FUNCTION_BLOCK TFModulePalletizer_Pinza_mag
VAR_INPUT
	Cmd 	: CommandBuffer;
	Cfg 	: Config;
	IN 		: TFMchinePalletizer_PinzaVentose_IN;
	IN_Ax 	: Module_Palletizer_Ax_IN;
	
	AspirazioneDX1 : POINTER TO TF_VacumOVEM;
	AspirazioneSX1 : POINTER TO TF_VacumOVEM;
	AspirazioneDX2 : POINTER TO TF_VacumOVEM;
	AspirazioneSX2 : POINTER TO TF_VacumOVEM;

	CilindroSbloccoRotazione 	: POINTER TO SC_Cylinder;
	CilindroSbloccoBascolante 	: POINTER TO SC_Cylinder;
	CilindroApertura 			: POINTER TO DC_Cylinder;
	
	ModuleJ : POINTER TO TFModulePalletizer_Ax;
	ModuleK : POINTER TO TFModulePalletizer_Ax;

	ManCmd 				: POINTER TO TFMachinePalletizer_PinzaVentoseManCmd;
	ElementoInPrelievo 	: TFMachinePalletizer_PlaceElement;
	DataElement			: TFMachinePalletizer_DataElement; (* Struttura dati che la macchina acquisisce/trasferisce in fase di pallettizzazione/depallettizazione *)
	PrelievoSuMagazino : BOOL;//indica che il prelievo è su cavallina

	Mission : POINTER TO TFMachinePalletizer_Mission;
	AbilitazioneSbloccoRotazione 	: BOOL;//Abilitazione sblocco rotazione pinza
	AbilitazioneSbloccoBascolante 	: BOOL;//Abilitazione sblocco bascolante pinza	
	IN_SimulazioneSenzaHW : BOOL;
	AbilitaAperturaAutomaticaPinza : BOOL;//Abilitazione apertura automatica pinza
END_VAR
VAR_OUTPUT
	CmdExe 		: CommandExe;
	CmdExd 		: CommandExe;
	CmdNext 	: Command;
	CmdLog 		: CommandLog;
	ProgramLog 	: ProgrammaLog; 
	State 		: State;
	StateLog 	: StateLog;
	Error 		: Error;
	ErrorLog 	: ErrorLog;
	Warning 	: Warning;
	WarningLog	: WarningLog;
	OUT 		: TFMachinePalletizer_PinzaVentose_OUT;
	StatoPinza 	: TFMachinePalletizer_PinzaState;

END_VAR
VAR
	Power 	: UINT;
	Init 	: BOOL;
	Timer 	: REAL;
	Timeout : REAL;
	TimerAspirazione 	: REAL;
	ParametersArray 	: ParametersArray;
	MAN_Actuator 		: UINT;
	MAN_Cmd 			: UINT;

	DistanzaFTC_J0 		: REAL;
	DistanzaFTC_J180 	: REAL;
	DistanzaFTC_K0 		: REAL;
	DistanzaFTC_K180 	: REAL;

	TimerPresaPiastrella : REAL;		
	DisattivazioneTotaleAspirazioni : bool;
	ByPassAttesaDistacco : BOOL;

	DistanzaJForzata : REAL;
	DistanzaKForzata : REAL;

END_VAR

IF NOT Init THEN
	TFCommandBufferClear(ADR(Cmd));
	TFCommandClear(ADR(CmdNext));
	TFCommandExeClear(ADR(CmdExe));
	TFStateUpdate(ADR(State),StateNOP);
	TFErrorClear(ADR(Error));
	TFWarningClear(ADR(Warning));
	Init := TRUE;
END_IF

(* Generic Timer - Add here all your Timers *)
TFTimerCall(ADR(Timer),Cfg.TimeBase);
TFTimerCall(ADR(Timeout),Cfg.TimeBase);
TFTimerCall(ADR(TimerPresaPiastrella),Cfg.TimeBase);
TFTimerCall(ADR(TimerAspirazione),Cfg.TimeBase);
(* External To Buffered Command *)
TFCommandToNext(ADR(Cmd),ADR(CmdNext),ADR(CmdExe),ADR(Cfg),ADR(Error),ADR(ErrorLog),ADR(State));

(* Buffered To Exe Command *)
TFCommandToExecution(ADR(CmdNext),ADR(CmdExe),ADR(Error),ADR(ErrorLog),ADR(State),ADR(CmdLog));

(* Chiamata FB *)
AspirazioneDX1^();
AspirazioneSX1^();
AspirazioneDX2^();
AspirazioneSX2^();
CilindroSbloccoRotazione^();
CilindroSbloccoBascolante^();

DistanzaFTC_J0 		:= Keyence_LRTB2000C(IN.InKeyence_J0_Byte0,IN.InKeyence_J0_Byte1);
DistanzaFTC_J180	:= Keyence_LRTB2000C(IN.InKeyence_J180_Byte0,IN.InKeyence_J180_Byte1);
DistanzaFTC_K0 		:= Keyence_LRTB2000C(IN.InKeyence_K0_Byte0,IN.InKeyence_K0_Byte1);
DistanzaFTC_K180	:= Keyence_LRTB2000C(IN.InKeyence_K180_Byte0,IN.InKeyence_K180_Byte1);

OUT.DistanzaFTC_J0 		:= DistanzaFTC_J0; 		
OUT.DistanzaFTC_J180	:= DistanzaFTC_J180;	
OUT.DistanzaFTC_K0 		:= DistanzaFTC_K0; 		
OUT.DistanzaFTC_K180   	:= DistanzaFTC_K180; 

DistanzaJForzata:=0;
IF ABS(DistanzaFTC_J0-DistanzaFTC_J180) > 30 THEN
	DistanzaJForzata := MIN(DistanzaFTC_J0,DistanzaFTC_J180);
END_IF
DistanzaKForzata:=0;
IF ABS(DistanzaFTC_K0-DistanzaFTC_K180) > 30 THEN
	DistanzaKForzata := MIN(DistanzaFTC_K0,DistanzaFTC_K180);
END_IF
OUT.DistanzaMedia := (DistanzaFTC_J0 + 	
                 DistanzaFTC_J180 +
                 DistanzaFTC_K0 + 	
                 DistanzaFTC_K180)/4;
				 
IF DistanzaKForzata > 0 THEN
	OUT.DistanzaMedia := (DistanzaJForzata +
                 DistanzaFTC_K0 + 	
                 DistanzaFTC_K180)/3;
END_IF
IF DistanzaJForzata > 0 THEN
	OUT.DistanzaMedia := (DistanzaFTC_J0 + 	
                 DistanzaFTC_J180 +
                 DistanzaKForzata)/3;
END_IF
IF DistanzaKForzata > 0 AND DistanzaJForzata > 0 THEN
	OUT.DistanzaMedia := (DistanzaJForzata +
                 DistanzaKForzata)/2;
END_IF

(* Exe Command *)
CASE CmdExe.Code OF

	(* ******************************************************************************************************** *)
	(* Nop  *)
	(* ******************************************************************************************************** *)
	CmdNOP:	;			
	(* ******************************************************************************************************** *)
	(* Stop *)
	(* ******************************************************************************************************** *)
	CmdSTOP:
		CASE CmdExe.CmdCase OF
			
			(* Case 0 *)
			0: 	TFStateUpdate(ADR(State),StateSTOP_RUN);
				TFTimerSet(ADR(Timeout),500,TRUE);
				TFCommandCase(ADR(CmdExe),1,CommandCase_INC);

			(* Case 1 - Clear All Commands*)
			1:	
				TFCommandCase(ADR(CmdExe),100,CommandCase_JMP);
			(* Case 100 *)
			100:TFStateUpdate(ADR(State),StateSTOP_END);
				TFCommandExeClear(ADR(CmdExe));

			ELSE
				TFError(ErrNOCMDCASE,ErrNULL,ADR(CmdExe),ADR(State),ADR(Error),ADR(ErrorLog));
		END_CASE;
	
	(* ******************************************************************************************************** *)
	(* Error Reset *)
	(* ******************************************************************************************************** *)
	CmdRESET:
		CASE CmdExe.CmdCase OF

			(* Case 0 *)
			0: 	TFStateUpdate(ADR(State),StateRESET_RUN);
				TFTimerSet(ADR(Timeout),2000+100,TRUE);
				TFTimerSet(ADR(Timer),2000,TRUE);
				TFCommandCase(ADR(CmdExe),1,CommandCase_JMP);

			
			(* Case 1 - RESET COMANDI*)
			1: 
				TFClearAllCmdModulePinzaMagazzino(AspirazioneDX1,AspirazioneSX1,AspirazioneDX2,AspirazioneSX2,CilindroSbloccoRotazione,CilindroSbloccoBascolante);
				TFCommandCase(ADR(CmdExe),1,CommandCase_INC);
			
			(* Case 2 - Invio comando di reset *)
			2:
				AspirazioneDX1^.Command^.ErrorReset 				:= TRUE;	
				AspirazioneSX1^.Command^.ErrorReset 				:= TRUE;	
				AspirazioneDX2^.Command^.ErrorReset 				:= TRUE;	
				AspirazioneSX2^.Command^.ErrorReset 				:= TRUE;	
				CilindroSbloccoRotazione^.Command.ErrorReset 	:= TRUE;	
				CilindroSbloccoBascolante^.Command.ErrorReset 	:= TRUE;	
				TFCommandCase(ADR(CmdExe),1,CommandCase_INC);
			
			(* Case 3 - Invio comando di reset *)
			3:
				IF (AspirazioneDX1^.Status.ErrorResetDone AND AspirazioneDX2^.Status.ErrorResetDone AND
					AspirazioneSX1^.Status.ErrorResetDone AND AspirazioneSX2^.Status.ErrorResetDone AND
					CilindroSbloccoRotazione^.Status.ErrorResetDone AND CilindroSbloccoBascolante^.Status.ErrorResetDone) OR IN_SimulazioneSenzaHW THEN					
					TFClearAllCmdModulePinzaMagazzino(AspirazioneDX1,AspirazioneSX1,AspirazioneDX2,AspirazioneSX2,CilindroSbloccoRotazione,CilindroSbloccoBascolante);
					TFCommandCase(ADR(CmdExe),99,CommandCase_JMP);
				ELSIF TFTimerDone(ADR(Timer)) THEN
					TFClearAllCmdModulePinzaMagazzino(AspirazioneDX1,AspirazioneSX1,AspirazioneDX2,AspirazioneSX2,CilindroSbloccoRotazione,CilindroSbloccoBascolante);
					TFError(ErrTORESET,ErrNULL,ADR(CmdExe),ADR(State),ADR(Error),ADR(ErrorLog));
				END_IF

			(* Case 99 *)
			99:	TFErrorClear(ADR(Error));
				TFWarningClear(ADR(Warning));
				TFCommandCase(ADR(CmdExe),100,CommandCase_JMP);

			(* Case 100 *)
			100:TFStateUpdate(ADR(State),StateRESET_END);
				TFCommandExeClear(ADR(CmdExe));

			ELSE
				TFError(ErrNOCMDCASE,ErrNULL,ADR(CmdExe),ADR(State),ADR(Error),ADR(ErrorLog));
		END_CASE;

		(*IF AspirazioneDX^.Status.ErrorID <> ErrNULL THEN
			TFClearAllCmdModulePinza(AspirazioneDX,AspirazioneSX,CilindroApertura,CilindroSbloccoRotazione,AspirazioneFaldaDX,AspirazioneFaldaSX,CilindroTasteggio);
			TFError(ErrCYLINDER,AspirazioneDX^.Status.ErrorID,ADR(CmdExe),ADR(State),ADR(Error),ADR(ErrorLog));
		ELSIF AspirazioneSX^.Status.ErrorID <> ErrNULL THEN
			TFClearAllCmdModulePinza(AspirazioneDX,AspirazioneSX,CilindroApertura,CilindroSbloccoRotazione,AspirazioneFaldaDX,AspirazioneFaldaSX,CilindroTasteggio);
			TFError(ErrCYLINDER,AspirazioneSX^.Status.ErrorID,ADR(CmdExe),ADR(State),ADR(Error),ADR(ErrorLog));
		ELSIF CilindroApertura^.Status.ErrorID <> ErrNULL THEN
			TFClearAllCmdModulePinza(AspirazioneDX,AspirazioneSX,CilindroApertura,CilindroSbloccoRotazione,AspirazioneFaldaDX,AspirazioneFaldaSX,CilindroTasteggio);
			TFError(ErrCYLINDER,CilindroApertura^.Status.ErrorID,ADR(CmdExe),ADR(State),ADR(Error),ADR(ErrorLog));
		ELSIF CilindroSbloccoRotazione^.Status.ErrorID <> ErrNULL THEN
			TFClearAllCmdModulePinza(AspirazioneDX,AspirazioneSX,CilindroApertura,CilindroSbloccoRotazione,AspirazioneFaldaDX,AspirazioneFaldaSX,CilindroTasteggio);
			TFError(ErrCYLINDER,CilindroSbloccoRotazione^.Status.ErrorID,ADR(CmdExe),ADR(State),ADR(Error),ADR(ErrorLog));
		ELSIF AspirazioneFaldaDX^.Status.ErrorID <> ErrNULL THEN
			TFClearAllCmdModulePinza(AspirazioneDX,AspirazioneSX,CilindroApertura,CilindroSbloccoRotazione,AspirazioneFaldaDX,AspirazioneFaldaSX,CilindroTasteggio);
			TFError(ErrCYLINDER,AspirazioneFaldaDX^.Status.ErrorID,ADR(CmdExe),ADR(State),ADR(Error),ADR(ErrorLog));
		ELSIF AspirazioneFaldaSX^.Status.ErrorID <> ErrNULL THEN
			TFClearAllCmdModulePinza(AspirazioneDX,AspirazioneSX,CilindroApertura,CilindroSbloccoRotazione,AspirazioneFaldaDX,AspirazioneFaldaSX,CilindroTasteggio);
			TFError(ErrCYLINDER,AspirazioneFaldaSX^.Status.ErrorID,ADR(CmdExe),ADR(State),ADR(Error),ADR(ErrorLog));
		*)
		IF TFTimerDone(ADR(Timeout)) THEN
			TFClearAllCmdModulePinzaMagazzino(AspirazioneDX1,AspirazioneSX1,AspirazioneDX2,AspirazioneSX2,CilindroSbloccoRotazione,CilindroSbloccoBascolante);
			TFError(ErrCMDTIMEOUT,ErrNULL,ADR(CmdExe),ADR(State),ADR(Error),ADR(ErrorLog));
		END_IF
	
	(* ******************************************************************************************************** *)
	(* Power *)
	(* ******************************************************************************************************** *)
	CmdPOWER:
		CASE CmdExe.CmdCase OF
			
			(* Case 0 *)
			0: 	TFStateUpdate(ADR(State),StatePOWER_RUN);
				TFTimerSet(ADR(Timeout),500,TRUE);
				TFCommandCase(ADR(CmdExe),100,CommandCase_JMP);

			1: TFCommandCase(ADR(CmdExe),100,CommandCase_JMP);
			(* Case 100 *)
			100:TFStateUpdate(ADR(State),StatePOWER_END);
				TFCommandExeClear(ADR(CmdExe));

			ELSE
				TFError(ErrNOCMDCASE,ErrNULL,ADR(CmdExe),ADR(State),ADR(Error),ADR(ErrorLog));
		END_CASE
	
	(* ******************************************************************************************************** *)
	(* Home *)
	(* ******************************************************************************************************** *)
	CmdHOME:
		CASE CmdExe.CmdCase OF

			(* Case 0 *)
			0: 	TFStateUpdate(ADR(State),StateHOME_RUN);
				TFTimerSet(ADR(Timeout),3000+200,TRUE);
				TFTimerSet(ADR(Timer),3000,TRUE);
				IF NOT IN_SimulazioneSenzaHW THEN
					TFCommandCase(ADR(CmdExe),1,CommandCase_INC);
				ELSE
					TFCommandCase(ADR(CmdExe),100,CommandCase_JMP);
				END_IF

			(* Case 1 - *)
			1: 
				TFCommandCase(ADR(CmdExe),10,CommandCase_JMP);

			(* Case 10 - Set automatico Soglie *)
			10:
				AspirazioneDX1^.Command^.Aspirazione_ON_ScritturaSoglia 	:= TRUE;
				AspirazioneSX1^.Command^.Aspirazione_ON_ScritturaSoglia 	:= TRUE;
				AspirazioneDX2^.Command^.Aspirazione_ON_ScritturaSoglia 	:= TRUE;
				AspirazioneSX2^.Command^.Aspirazione_ON_ScritturaSoglia 	:= TRUE;
				IF AspirazioneDX1^.Status.CommandDone AND AspirazioneSX1^.Status.CommandDone AND
					AspirazioneDX2^.Status.CommandDone AND AspirazioneSX2^.Status.CommandDone THEN
						TFClearAllCmdModulePinzaMagazzino(AspirazioneDX1,AspirazioneSX1,AspirazioneDX2,AspirazioneSX2,CilindroSbloccoRotazione,CilindroSbloccoBascolante);
						TFCommandCase(ADR(CmdExe),100,CommandCase_JMP);
				ELSIF TFTimerDone(ADR(Timer)) THEN
					TFClearAllCmdModulePinzaMagazzino(AspirazioneDX1,AspirazioneSX1,AspirazioneDX2,AspirazioneSX2,CilindroSbloccoRotazione,CilindroSbloccoBascolante);
					TFError(ErrTOHOME,ErrNULL,ADR(CmdExe),ADR(State),ADR(Error),ADR(ErrorLog));
				END_IF
			
	
			(* Case 100 *)
			100:TFStateUpdate(ADR(State),StateHOME_END);
				TFCommandExeClear(ADR(CmdExe));

			ELSE
				TFError(ErrNOCMDCASE,ErrNULL,ADR(CmdExe),ADR(State),ADR(Error),ADR(ErrorLog));
		END_CASE;
		
		IF AspirazioneDX1^.Status.ErrorID <> ErrNULL AND NOT IN_SimulazioneSenzaHW THEN
			TFClearAllCmdModulePinzaMagazzino(AspirazioneDX1,AspirazioneSX1,AspirazioneDX2,AspirazioneSX2,CilindroSbloccoRotazione,CilindroSbloccoBascolante);
			TFError(ErrCYLINDER,AspirazioneDX1^.Status.ErrorID,ADR(CmdExe),ADR(State),ADR(Error),ADR(ErrorLog));
		ELSIF AspirazioneSX1^.Status.ErrorID <> ErrNULL AND NOT IN_SimulazioneSenzaHW THEN
			TFClearAllCmdModulePinzaMagazzino(AspirazioneDX1,AspirazioneSX1,AspirazioneDX2,AspirazioneSX2,CilindroSbloccoRotazione,CilindroSbloccoBascolante);
			TFError(ErrCYLINDER,AspirazioneSX1^.Status.ErrorID,ADR(CmdExe),ADR(State),ADR(Error),ADR(ErrorLog));
		ELSIF AspirazioneDX2^.Status.ErrorID <> ErrNULL AND NOT IN_SimulazioneSenzaHW THEN
			TFClearAllCmdModulePinzaMagazzino(AspirazioneDX1,AspirazioneSX1,AspirazioneDX2,AspirazioneSX2,CilindroSbloccoRotazione,CilindroSbloccoBascolante);
			TFError(ErrCYLINDER,AspirazioneDX2^.Status.ErrorID,ADR(CmdExe),ADR(State),ADR(Error),ADR(ErrorLog));
		ELSIF AspirazioneSX2^.Status.ErrorID <> ErrNULL AND NOT IN_SimulazioneSenzaHW THEN
			TFClearAllCmdModulePinzaMagazzino(AspirazioneDX1,AspirazioneSX1,AspirazioneDX2,AspirazioneSX2,CilindroSbloccoRotazione,CilindroSbloccoBascolante);
			TFError(ErrCYLINDER,AspirazioneSX2^.Status.ErrorID,ADR(CmdExe),ADR(State),ADR(Error),ADR(ErrorLog));
		ELSIF CilindroSbloccoRotazione^.Status.ErrorID <> ErrNULL THEN
			TFClearAllCmdModulePinzaMagazzino(AspirazioneDX1,AspirazioneSX1,AspirazioneDX2,AspirazioneSX2,CilindroSbloccoRotazione,CilindroSbloccoBascolante);
			TFError(ErrCYLINDER,CilindroSbloccoRotazione^.Status.ErrorID,ADR(CmdExe),ADR(State),ADR(Error),ADR(ErrorLog));
		ELSIF TFTimerDone(ADR(Timeout)) THEN
			TFClearAllCmdModulePinzaMagazzino(AspirazioneDX1,AspirazioneSX1,AspirazioneDX2,AspirazioneSX2,CilindroSbloccoRotazione,CilindroSbloccoBascolante);
			TFError(ErrCMDTIMEOUT,ErrNULL,ADR(CmdExe),ADR(State),ADR(Error),ADR(ErrorLog));
		END_IF

	(* ******************************************************************************************************** *)
	(* Manual *)
	(* ******************************************************************************************************** *)
	CmdMAN:
		CASE CmdExe.CmdCase OF
			(* Case 0 *)
			0: 	TFStateUpdate(ADR(State),StateMAN_RUN);
				TFTimerSet(ADR(Timeout),3000,TRUE);
				TFTimerSet(ADR(Timer),10,TRUE);
				IF TFCommandParRead(CmdExe.Cmd.Parameter,ADR(ParametersArray),2) THEN
					MAN_Actuator	:= STRING_TO_UINT(ParametersArray.Parameters[0]);
					MAN_Cmd		:= STRING_TO_UINT(ParametersArray.Parameters[1]);
				ELSE
					TFError(ErrCMDPARNUM,ErrNULL,ADR(CmdExe),ADR(State),ADR(Error),ADR(ErrorLog));
					RETURN;
				END_IF;

				CASE MAN_Actuator OF
					(* Case 0..99 for Actuators *)
					(* Case 100..199  for Axis *)

					(* Case Nop *)
					0:	;

					(* Case 1: *)
					1:	CASE MAN_Cmd OF
							0:	;
							
							
							(* Case 20: Sgancio Sblocco Rotazione *)
							20:	
								CilindroSbloccoRotazione^.Command.Activation 	:= TRUE;
								CilindroSbloccoRotazione^.Command.Deactivation 	:= FALSE;
								TFTimerSet(ADR(Timeout),3000,TRUE);
								TFCommandCase(ADR(CmdExe),20,CommandCase_JMP);
								
							(* Case 21: Aggancio Sblocco Rotazione *)
							21:	
								CilindroSbloccoRotazione^.Command.Activation 	:= FALSE;
								CilindroSbloccoRotazione^.Command.Deactivation 	:= TRUE;
								TFTimerSet(ADR(Timeout),3000,TRUE);
								TFCommandCase(ADR(CmdExe),20,CommandCase_JMP);
	
							(* Case 50: Ativazione Aspirazione SX *)
							50:	
								
								IF NOT IN_SimulazioneSenzaHW THEN 
									AspirazioneSX1^.Command^.Aspirazione_ON		:= TRUE;
									AspirazioneSX1^.Command^.Aspirazione_OFF 	:= FALSE;
									AspirazioneDX1^.Command^.Aspirazione_ON 	:= TRUE;
									AspirazioneDX1^.Command^.Aspirazione_OFF 	:= FALSE;
									AspirazioneSX2^.Command^.Aspirazione_ON 	:= TRUE;
									AspirazioneSX2^.Command^.Aspirazione_OFF 	:= FALSE;
									AspirazioneDX2^.Command^.Aspirazione_ON 	:= TRUE;
									AspirazioneDX2^.Command^.Aspirazione_OFF 	:= FALSE;
	
									TFTimerSet(ADR(Timeout),3000,TRUE);
									TFCommandCase(ADR(CmdExe),50,CommandCase_JMP);
								ELSE
									TFCommandCase(ADR(CmdExe),1,CommandCase_JMP);
								END_IF
										
							(* Case 51: Disattivazione Aspirazione SX *)
							51:	
								StatoPinza.ElementoPrelevato := FALSE;
								IF NOT IN_SimulazioneSenzaHW THEN 
									AspirazioneSX1^.Command^.Aspirazione_ON 	:= FALSE;
									AspirazioneSX1^.Command^.Aspirazione_OFF 	:= TRUE;
									AspirazioneDX1^.Command^.Aspirazione_ON 	:= FALSE;
									AspirazioneDX1^.Command^.Aspirazione_OFF 	:= TRUE;
									AspirazioneSX2^.Command^.Aspirazione_ON 	:= FALSE;
									AspirazioneSX2^.Command^.Aspirazione_OFF 	:= TRUE;
									AspirazioneDX2^.Command^.Aspirazione_ON 	:= FALSE;
									AspirazioneDX2^.Command^.Aspirazione_OFF 	:= TRUE;
									TFTimerSet(ADR(Timeout),3000,TRUE);
									TFCommandCase(ADR(CmdExe),50,CommandCase_JMP);
								ELSE
									TFCommandCase(ADR(CmdExe),1,CommandCase_JMP);
								END_IF

							(* Case 60: Ativazione Aspirazione DX *)
							60:	
								IF NOT IN_SimulazioneSenzaHW THEN 
									AspirazioneSX1^.Command^.Aspirazione_ON 	:= TRUE;
									AspirazioneSX1^.Command^.Aspirazione_OFF 	:= FALSE;
									AspirazioneDX1^.Command^.Aspirazione_ON 	:= TRUE;
									AspirazioneDX1^.Command^.Aspirazione_OFF 	:= FALSE;
									AspirazioneSX2^.Command^.Aspirazione_ON 	:= TRUE;
									AspirazioneSX2^.Command^.Aspirazione_OFF 	:= FALSE;
									AspirazioneDX2^.Command^.Aspirazione_ON 	:= TRUE;
									AspirazioneDX2^.Command^.Aspirazione_OFF 	:= FALSE;
									TFTimerSet(ADR(Timeout),3000,TRUE);
									TFCommandCase(ADR(CmdExe),60,CommandCase_JMP);
								ELSE
									TFCommandCase(ADR(CmdExe),1,CommandCase_JMP);
								END_IF

							(* Case 61: Disattivazione Aspirazione SX *)
							61:	
								StatoPinza.ElementoPrelevato := FALSE;
								IF NOT IN_SimulazioneSenzaHW THEN 
									AspirazioneDX1^.Command^.Aspirazione_ON  := FALSE;
									AspirazioneDX1^.Command^.Aspirazione_OFF := TRUE;
									AspirazioneSX1^.Command^.Aspirazione_ON  := FALSE;
									AspirazioneSX1^.Command^.Aspirazione_OFF := TRUE;
									AspirazioneDX2^.Command^.Aspirazione_ON  := FALSE;
									AspirazioneDX2^.Command^.Aspirazione_OFF := TRUE;
									AspirazioneSX2^.Command^.Aspirazione_ON  := FALSE;
									AspirazioneSX2^.Command^.Aspirazione_OFF := TRUE;
									StatoPinza.ElementoPrelevato := FALSE;
									TFTimerSet(ADR(Timeout),3000,TRUE);
									TFCommandCase(ADR(CmdExe),60,CommandCase_JMP);
								ELSE
									TFCommandCase(ADR(CmdExe),1,CommandCase_JMP);
								END_IF
							ELSE
								TFError(ErrNOCMDCASE,ErrNULL,ADR(CmdExe),ADR(State),ADR(Error),ADR(ErrorLog));
						END_CASE;

					100:CASE MAN_Cmd OF
							0:	;
							ELSE
								TFError(ErrNOCMDCASE,ErrNULL,ADR(CmdExe),ADR(State),ADR(Error),ADR(ErrorLog));
						END_CASE;

					ELSE
						TFError(ErrNOCMDCASE,ErrNULL,ADR(CmdExe),ADR(State),ADR(Error),ADR(ErrorLog));
				END_CASE;

				//IF CmdExe.CmdCase = 0 THEN
					//TFCommandCase(ADR(CmdExe),1,CommandCase_INC);
				//END_IF

			(* Case 1 - *)
			1: 	IF (MAN_Cmd = 0) OR TFTimerDone(ADR(Timer)) THEN
					(* Clear All Output Here *)
					;
					TFStateUpdate(ADR(State),StateMAN_END);
					TFCommandExeClear(ADR(CmdExe));
				END_IF;

			(* Case 20 - CilindroSbloccoRotazione *)
			20: 
				IF CilindroSbloccoRotazione^.Status.Inactive AND CilindroSbloccoRotazione^.Command.Deactivation OR
					CilindroSbloccoRotazione^.Status.Active AND CilindroSbloccoRotazione^.Command.Activation THEN
						CilindroSbloccoRotazione^.Command.Activation 	:= FALSE;
						CilindroSbloccoRotazione^.Command.Deactivation 	:= FALSE;
						TFCommandCase(ADR(CmdExe),100,CommandCase_JMP);
				ELSIF CilindroSbloccoRotazione^.Status.ErrorID <> ErrNULL THEN
					TFClearAllCmdModulePinzaMagazzino(AspirazioneDX1,AspirazioneSX1,AspirazioneDX2,AspirazioneSX2,CilindroSbloccoRotazione,CilindroSbloccoBascolante);
					TFError(ErrCYLINDER,CilindroSbloccoRotazione^.Status.ErrorID,ADR(CmdExe),ADR(State),ADR(Error),ADR(ErrorLog));
				END_IF

			(* Case 50 - AspirazioneSX *)
			50: 
				IF AspirazioneSX1^.Status.CommandDone AND AspirazioneDX1^.Status.CommandDone AND
					AspirazioneSX2^.Status.CommandDone AND AspirazioneDX2^.Status.CommandDone THEN
						TFClearAllCmdModulePinzaMagazzino(AspirazioneDX1,AspirazioneSX1,AspirazioneDX2,AspirazioneSX2,CilindroSbloccoRotazione,CilindroSbloccoBascolante);
						TFCommandCase(ADR(CmdExe),100,CommandCase_JMP);
				ELSIF AspirazioneSX1^.Status.ErrorID <> ErrNULL THEN
					TFClearAllCmdModulePinzaMagazzino(AspirazioneDX1,AspirazioneSX1,AspirazioneDX2,AspirazioneSX2,CilindroSbloccoRotazione,CilindroSbloccoBascolante);
					TFError(ErrCYLINDER,AspirazioneSX1^.Status.ErrorID,ADR(CmdExe),ADR(State),ADR(Error),ADR(ErrorLog));
				ELSIF AspirazioneDX1^.Status.ErrorID <> ErrNULL THEN
					TFClearAllCmdModulePinzaMagazzino(AspirazioneDX1,AspirazioneSX1,AspirazioneDX2,AspirazioneSX2,CilindroSbloccoRotazione,CilindroSbloccoBascolante);
					TFError(ErrCYLINDER,AspirazioneDX1^.Status.ErrorID,ADR(CmdExe),ADR(State),ADR(Error),ADR(ErrorLog));
				ELSIF AspirazioneSX2^.Status.ErrorID <> ErrNULL THEN
					TFClearAllCmdModulePinzaMagazzino(AspirazioneDX1,AspirazioneSX1,AspirazioneDX2,AspirazioneSX2,CilindroSbloccoRotazione,CilindroSbloccoBascolante);
					TFError(ErrCYLINDER,AspirazioneSX2^.Status.ErrorID,ADR(CmdExe),ADR(State),ADR(Error),ADR(ErrorLog));
				ELSIF AspirazioneDX2^.Status.ErrorID <> ErrNULL THEN
					TFClearAllCmdModulePinzaMagazzino(AspirazioneDX1,AspirazioneSX1,AspirazioneDX2,AspirazioneSX2,CilindroSbloccoRotazione,CilindroSbloccoBascolante);
					TFError(ErrCYLINDER,AspirazioneDX2^.Status.ErrorID,ADR(CmdExe),ADR(State),ADR(Error),ADR(ErrorLog));
				END_IF

			(* Case 60 - AspirazioneDX *)
			60: 
				IF AspirazioneSX1^.Status.CommandDone AND AspirazioneDX1^.Status.CommandDone AND
					AspirazioneSX2^.Status.CommandDone AND AspirazioneDX2^.Status.CommandDone THEN
						TFClearAllCmdModulePinzaMagazzino(AspirazioneDX1,AspirazioneSX1,AspirazioneDX2,AspirazioneSX2,CilindroSbloccoRotazione,CilindroSbloccoBascolante);
						TFCommandCase(ADR(CmdExe),100,CommandCase_JMP);
				ELSIF AspirazioneSX1^.Status.ErrorID <> ErrNULL THEN
					TFClearAllCmdModulePinzaMagazzino(AspirazioneDX1,AspirazioneSX1,AspirazioneDX2,AspirazioneSX2,CilindroSbloccoRotazione,CilindroSbloccoBascolante);
					TFError(ErrCYLINDER,AspirazioneSX1^.Status.ErrorID,ADR(CmdExe),ADR(State),ADR(Error),ADR(ErrorLog));
				ELSIF AspirazioneDX1^.Status.ErrorID <> ErrNULL THEN
					TFClearAllCmdModulePinzaMagazzino(AspirazioneDX1,AspirazioneSX1,AspirazioneDX2,AspirazioneSX2,CilindroSbloccoRotazione,CilindroSbloccoBascolante);
					TFError(ErrCYLINDER,AspirazioneDX1^.Status.ErrorID,ADR(CmdExe),ADR(State),ADR(Error),ADR(ErrorLog));
				ELSIF AspirazioneSX2^.Status.ErrorID <> ErrNULL THEN
					TFClearAllCmdModulePinzaMagazzino(AspirazioneDX1,AspirazioneSX1,AspirazioneDX2,AspirazioneSX2,CilindroSbloccoRotazione,CilindroSbloccoBascolante);
					TFError(ErrCYLINDER,AspirazioneSX2^.Status.ErrorID,ADR(CmdExe),ADR(State),ADR(Error),ADR(ErrorLog));
				ELSIF AspirazioneDX2^.Status.ErrorID <> ErrNULL THEN
					TFClearAllCmdModulePinzaMagazzino(AspirazioneDX1,AspirazioneSX1,AspirazioneDX2,AspirazioneSX2,CilindroSbloccoRotazione,CilindroSbloccoBascolante);
					TFError(ErrCYLINDER,AspirazioneDX2^.Status.ErrorID,ADR(CmdExe),ADR(State),ADR(Error),ADR(ErrorLog));
				END_IF

			(* Case 100 - End *)
			100:(* Clear All Output Here *)
				TFStateUpdate(ADR(State),StateMAN_END);
				TFCommandExeClear(ADR(CmdExe));

			ELSE
				TFError(ErrNOCMDCASE,ErrNULL,ADR(CmdExe),ADR(State),ADR(Error),ADR(ErrorLog));
		END_CASE;

		IF TFTimerDone(ADR(Timeout)) THEN
			TFClearAllCmdModulePinzaMagazzino(AspirazioneDX1,AspirazioneSX1,AspirazioneDX2,AspirazioneSX2,CilindroSbloccoRotazione,CilindroSbloccoBascolante);
			TFError(ErrCMDTIMEOUT,ErrNULL,ADR(CmdExe),ADR(State),ADR(Error),ADR(ErrorLog));
		END_IF
	

	(* ******************************************************************************************************** *)
	(* PRELOAD - Attivazione vuoto *)
	(* ******************************************************************************************************** *)
	CmdPRELOAD:
		CASE CmdExe.CmdCase OF
			
			(* Case 0 - Init Command*)
			0: 	TFStateUpdate(ADR(State),StatePRELOAD_RUN);
				TFTimerSet(ADR(Timeout),30000+200,TRUE);
				TFTimerSet(ADR(Timer),30000,TRUE);
				PrelievoSuMagazino := FALSE;
				StatoPinza.ElementoPrelevato := FALSE;
				IF TFCommandParRead(CmdExe.Cmd.Parameter,ADR(ParametersArray),1) THEN
					PrelievoSuMagazino	:= STRING_TO_BOOL(ParametersArray.Parameters[0]);
					IF NOT IN_SimulazioneSenzaHW THEN
						TFCommandCase(ADR(CmdExe),40,CommandCase_JMP);
					ELSE
						TFCommandCase(ADR(CmdExe),100,CommandCase_JMP);
					END_IF
				ELSE
					TFError(ErrCMDPARNUM,ErrNULL,ADR(CmdExe),ADR(State),ADR(Error),ADR(ErrorLog));
					RETURN;
				END_IF;
				
			(* Case 10 - CilindroSbloccoRotazione *)
			10: 
				IF PrelievoSuMagazino AND FALSE THEN
					CilindroSbloccoRotazione^.Command.Activation 	:= AbilitazioneSbloccoRotazione;
					CilindroSbloccoRotazione^.Command.Deactivation 	:= FALSE;
	
					IF (CilindroSbloccoRotazione^.Status.Active OR NOT AbilitazioneSbloccoRotazione)THEN
						CilindroSbloccoRotazione^.Command.Activation 	:= FALSE;
						CilindroSbloccoRotazione^.Command.Deactivation 	:= FALSE;
						TFCommandCase(ADR(CmdExe),40,CommandCase_JMP);
					ELSIF CilindroSbloccoRotazione^.Status.ErrorID <> ErrNULL AND AbilitazioneSbloccoRotazione THEN
						TFClearAllCmdModulePinzaMagazzino(AspirazioneDX1,AspirazioneSX1,AspirazioneDX2,AspirazioneSX2,CilindroSbloccoRotazione,CilindroSbloccoBascolante);
						TFError(ErrCYLINDER,CilindroSbloccoRotazione^.Status.ErrorID,ADR(CmdExe),ADR(State),ADR(Error),ADR(ErrorLog));
					END_IF
				ELSE
					TFCommandCase(ADR(CmdExe),40,CommandCase_JMP);
				END_IF


			(* Case 40 - AspirazioneDX + AspirazioneSX *)
			40: 
				AspirazioneDX1^.Command^.Aspirazione_ON 	:= TRUE;
				AspirazioneDX1^.Command^.Aspirazione_OFF 	:= FALSE;
				AspirazioneSX1^.Command^.Aspirazione_ON 	:= TRUE;
				AspirazioneSX1^.Command^.Aspirazione_OFF 	:= FALSE;
				AspirazioneDX2^.Command^.Aspirazione_ON 	:= TRUE;
				AspirazioneDX2^.Command^.Aspirazione_OFF 	:= FALSE;
				AspirazioneSX2^.Command^.Aspirazione_ON 	:= TRUE;
				AspirazioneSX2^.Command^.Aspirazione_OFF 	:= FALSE;
	
				IF (AspirazioneDX1^.Status.CommandDone AND AspirazioneSX1^.Status.CommandDone AND
					AspirazioneDX2^.Status.CommandDone AND AspirazioneSX2^.Status.CommandDone) OR IN.ByPassSensoreVuoto THEN
						TFClearAllCmdModulePinzaMagazzino(AspirazioneDX1,AspirazioneSX1,AspirazioneDX2,AspirazioneSX2,CilindroSbloccoRotazione,CilindroSbloccoBascolante);
						TFCommandCase(ADR(CmdExe),100,CommandCase_JMP);
				ELSIF AspirazioneSX1^.Status.ErrorID <> ErrNULL AND NOT IN_SimulazioneSenzaHW THEN
					TFClearAllCmdModulePinzaMagazzino(AspirazioneDX1,AspirazioneSX1,AspirazioneDX2,AspirazioneSX2,CilindroSbloccoRotazione,CilindroSbloccoBascolante);
					TFError(ErrCYLINDER,AspirazioneSX1^.Status.ErrorID,ADR(CmdExe),ADR(State),ADR(Error),ADR(ErrorLog));
				ELSIF AspirazioneDX1^.Status.ErrorID <> ErrNULL AND NOT IN_SimulazioneSenzaHW THEN
					TFClearAllCmdModulePinzaMagazzino(AspirazioneDX1,AspirazioneSX1,AspirazioneDX2,AspirazioneSX2,CilindroSbloccoRotazione,CilindroSbloccoBascolante);
					TFError(ErrCYLINDER,AspirazioneDX1^.Status.ErrorID,ADR(CmdExe),ADR(State),ADR(Error),ADR(ErrorLog));
				ELSIF AspirazioneSX2^.Status.ErrorID <> ErrNULL THEN
					TFClearAllCmdModulePinzaMagazzino(AspirazioneDX1,AspirazioneSX1,AspirazioneDX2,AspirazioneSX2,CilindroSbloccoRotazione,CilindroSbloccoBascolante);
					TFError(ErrCYLINDER,AspirazioneSX2^.Status.ErrorID,ADR(CmdExe),ADR(State),ADR(Error),ADR(ErrorLog));
				ELSIF AspirazioneDX2^.Status.ErrorID <> ErrNULL THEN
					TFClearAllCmdModulePinzaMagazzino(AspirazioneDX1,AspirazioneSX1,AspirazioneDX2,AspirazioneSX2,CilindroSbloccoRotazione,CilindroSbloccoBascolante);
					TFError(ErrCYLINDER,AspirazioneDX2^.Status.ErrorID,ADR(CmdExe),ADR(State),ADR(Error),ADR(ErrorLog));
				END_IF
				
			(* Case 100 *)
			100:TFStateUpdate(ADR(State),StatePRELOAD_END);
				TFCommandExeClear(ADR(CmdExe));

			ELSE
				TFError(ErrNOCMDCASE,ErrNULL,ADR(CmdExe),ADR(State),ADR(Error),ADR(ErrorLog));
		END_CASE

		IF TFTimerDone(ADR(Timeout)) THEN
			TFClearAllCmdModulePinzaMagazzino(AspirazioneDX1,AspirazioneSX1,AspirazioneDX2,AspirazioneSX2,CilindroSbloccoRotazione,CilindroSbloccoBascolante);
			TFError(ErrCMDTIMEOUT,ErrNULL,ADR(CmdExe),ADR(State),ADR(Error),ADR(ErrorLog));
		END_IF
	
	(* ******************************************************************************************************** *)
	(* LOAD - Presa del pezzo *)
	(* ******************************************************************************************************** *)
	CmdCHECKPRESENCE:
		CASE CmdExe.CmdCase OF
			
			(* Case 0 - Init Command*)
			0: 	TFStateUpdate(ADR(State),StateCHECKPRESENCE_RUN);
				TFTimerSet(ADR(Timeout),60000.0+100+HMI_TempoControlloPresaPiastrella,TRUE);
				TFTimerSet(ADR(Timer),2000.0+HMI_TempoControlloPresaPiastrella,TRUE);
				TFTimerSet(ADR(TimerPresaPiastrella),HMI_TempoControlloPresaPiastrella,TRUE);
				StatoPinza.ElementoPrelevato := FALSE;

				TFCommandCase(ADR(CmdExe),1,CommandCase_INC);
				
			(* Case 1 - *)					
			1:
				IF IN.ByPassSensoreVuoto OR TFTimerDone(ADR(TimerPresaPiastrella)) THEN 
					//Tutte piastrelle o tutte falde
					IF (AspirazioneDX1^.Status.DepressioneSoglia1_OK AND AspirazioneSX1^.Status.DepressioneSoglia1_OK AND
						 AspirazioneDX2^.Status.DepressioneSoglia1_OK AND AspirazioneSX2^.Status.DepressioneSoglia1_OK) OR IN.ByPassSensoreVuoto THEN
						StatoPinza.ElementoPrelevato := TRUE;
						TFCommandCase(ADR(CmdExe),11,CommandCase_JMP);
					ELSIF TFTimerDone(ADR(TimerPresaPiastrella)) THEN
						TFCommandCase(ADR(CmdExe),11,CommandCase_JMP);
						StatoPinza.ElementoPrelevato := IN.ByPassSensoreVuoto;	
					END_IF			
				END_IF
				IF TFTimerDone(ADR(Timer)) THEN
					TFClearAllCmdModulePinzaMagazzino(AspirazioneDX1,AspirazioneSX1,AspirazioneDX2,AspirazioneSX2,CilindroSbloccoRotazione,CilindroSbloccoBascolante);
					TFError(ErrMalfunzionamentoSensoriPresenzaPinza,ErrNULL,ADR(CmdExe),ADR(State),ADR(Error),ADR(ErrorLog));
				ELSIF TFTimerDone(ADR(Timeout)) THEN
					TFClearAllCmdModulePinzaMagazzino(AspirazioneDX1,AspirazioneSX1,AspirazioneDX2,AspirazioneSX2,CilindroSbloccoRotazione,CilindroSbloccoBascolante);
					TFError(ErrCMDTIMEOUT,ErrNULL,ADR(CmdExe),ADR(State),ADR(Error),ADR(ErrorLog));
				END_IF
						
			(* Case 11 - *)		
			11:
				TFStateUpdate(ADR(State),StateCHECKPRESENCE_RUN+10);
				TFCommandCase(ADR(CmdExe),100,CommandCase_JMP);
								
					
			(* Case 100 *)
			100:TFStateUpdate(ADR(State),StateCHECKPRESENCE_END);
				TFCommandExeClear(ADR(CmdExe));

			ELSE
				TFError(ErrNOCMDCASE,ErrNULL,ADR(CmdExe),ADR(State),ADR(Error),ADR(ErrorLog));
		END_CASE

	(* ******************************************************************************************************** *)
	(* CmdSbloccaBascolante - SGANCIO BASCULANTE *)
	(* ******************************************************************************************************** *)
	CmdSbloccaBascolante:
		CASE CmdExe.CmdCase OF
			
			(* Case 0 - Init Command*)
			0: 	TFStateUpdate(ADR(State),StateSbloccaBascolante_RUN);
				TFTimerSet(ADR(Timeout),30000+200,TRUE);
				TFTimerSet(ADR(Timer),30000,TRUE);
				IF NOT IN_SimulazioneSenzaHW THEN
					TFCommandCase(ADR(CmdExe),10,CommandCase_JMP);
				ELSE
					TFCommandCase(ADR(CmdExe),100,CommandCase_JMP);
				END_IF
				
			(* Case 10 - CilindroSblocco bacolante *)
			10: 
				CilindroSbloccoBascolante^.Command.Activation 	:= AbilitazioneSbloccoBascolante;
				CilindroSbloccoBascolante^.Command.Deactivation := FALSE;

				IF (CilindroSbloccoBascolante^.Status.Active OR NOT AbilitazioneSbloccoBascolante)THEN
					CilindroSbloccoBascolante^.Command.Activation 	:= FALSE;
					CilindroSbloccoBascolante^.Command.Deactivation 	:= FALSE;
					TFCommandCase(ADR(CmdExe),100,CommandCase_JMP);
				ELSIF CilindroSbloccoBascolante^.Status.ErrorID <> ErrNULL AND AbilitazioneSbloccoBascolante THEN
					TFClearAllCmdModulePinzaMagazzino(AspirazioneDX1,AspirazioneSX1,AspirazioneDX2,AspirazioneSX2,CilindroSbloccoRotazione,CilindroSbloccoBascolante);
					TFError(ErrCYLINDER,CilindroSbloccoBascolante^.Status.ErrorID,ADR(CmdExe),ADR(State),ADR(Error),ADR(ErrorLog));
				END_IF

				
			(* Case 100 *)
			100:TFStateUpdate(ADR(State),StateSbloccaBascolante_END);
				TFCommandExeClear(ADR(CmdExe));

			ELSE
				TFError(ErrNOCMDCASE,ErrNULL,ADR(CmdExe),ADR(State),ADR(Error),ADR(ErrorLog));
		END_CASE

		IF TFTimerDone(ADR(Timeout)) THEN
			TFClearAllCmdModulePinzaMagazzino(AspirazioneDX1,AspirazioneSX1,AspirazioneDX2,AspirazioneSX2,CilindroSbloccoRotazione,CilindroSbloccoBascolante);
			TFError(ErrCMDTIMEOUT,ErrNULL,ADR(CmdExe),ADR(State),ADR(Error),ADR(ErrorLog));
		END_IF
		
		(* ******************************************************************************************************** *)
	(* CmdBloccaBascolante - AGGANCIO BASCULANTE *)
	(* ******************************************************************************************************** *)
	CmdBloccaBascolante:
		CASE CmdExe.CmdCase OF
			
			(* Case 0 - Init Command*)
			0: 	TFStateUpdate(ADR(State),StateBloccaBascolante_RUN);
				TFTimerSet(ADR(Timeout),30000+200,TRUE);
				TFTimerSet(ADR(Timer),30000,TRUE);
				IF NOT IN_SimulazioneSenzaHW THEN
					TFCommandCase(ADR(CmdExe),10,CommandCase_JMP);
				ELSE
					TFCommandCase(ADR(CmdExe),100,CommandCase_JMP);
				END_IF
				
			(* Case 10 - CilindroSblocco bacolante *)
			10: 
				CilindroSbloccoBascolante^.Command.Activation 	:= FALSE;
				CilindroSbloccoBascolante^.Command.Deactivation := TRUE;

				IF  CilindroSbloccoBascolante^.Status.Inactive THEN
					CilindroSbloccoBascolante^.Command.Activation 	:= FALSE;
					CilindroSbloccoBascolante^.Command.Deactivation := FALSE;
					TFCommandCase(ADR(CmdExe),100,CommandCase_JMP);
				ELSIF CilindroSbloccoBascolante^.Status.ErrorID <> ErrNULL AND AbilitazioneSbloccoBascolante THEN
					TFClearAllCmdModulePinzaMagazzino(AspirazioneDX1,AspirazioneSX1,AspirazioneDX2,AspirazioneSX2,CilindroSbloccoRotazione,CilindroSbloccoBascolante);
					TFError(ErrCYLINDER,CilindroSbloccoBascolante^.Status.ErrorID,ADR(CmdExe),ADR(State),ADR(Error),ADR(ErrorLog));
				END_IF

				
			(* Case 100 *)
			100:TFStateUpdate(ADR(State),StateBloccaBascolante_END);
				TFCommandExeClear(ADR(CmdExe));

			ELSE
				TFError(ErrNOCMDCASE,ErrNULL,ADR(CmdExe),ADR(State),ADR(Error),ADR(ErrorLog));
		END_CASE

		IF TFTimerDone(ADR(Timeout)) THEN
			TFClearAllCmdModulePinzaMagazzino(AspirazioneDX1,AspirazioneSX1,AspirazioneDX2,AspirazioneSX2,CilindroSbloccoRotazione,CilindroSbloccoBascolante);
			TFError(ErrCMDTIMEOUT,ErrNULL,ADR(CmdExe),ADR(State),ADR(Error),ADR(ErrorLog));
		END_IF
		
	(* ******************************************************************************************************** *)
	(* CmdSbloccaRotazione - SGANCIO rotazione *)
	(* ******************************************************************************************************** *)
	CmdSbloccaRotazione:
		CASE CmdExe.CmdCase OF
			
			(* Case 0 - Init Command*)
			0: 	TFStateUpdate(ADR(State),StateSbloccaRotazione_RUN);
				TFTimerSet(ADR(Timeout),30000+200,TRUE);
				TFTimerSet(ADR(Timer),30000,TRUE);
				IF NOT IN_SimulazioneSenzaHW THEN
					TFCommandCase(ADR(CmdExe),10,CommandCase_JMP);
				ELSE
					TFCommandCase(ADR(CmdExe),100,CommandCase_JMP);
				END_IF
				
			(* Case 10 - CilindroSblocco bacolante *)
			10: 
				CilindroSbloccoRotazione^.Command.Activation 	:= AbilitazioneSbloccoRotazione;
				CilindroSbloccoRotazione^.Command.Deactivation := FALSE;

				IF (CilindroSbloccoRotazione^.Status.Active OR NOT AbilitazioneSbloccoRotazione)THEN
					CilindroSbloccoRotazione^.Command.Activation 	:= FALSE;
					CilindroSbloccoRotazione^.Command.Deactivation 	:= FALSE;
					TFCommandCase(ADR(CmdExe),100,CommandCase_JMP);
				ELSIF CilindroSbloccoBascolante^.Status.ErrorID <> ErrNULL AND AbilitazioneSbloccoRotazione THEN
					TFClearAllCmdModulePinzaMagazzino(AspirazioneDX1,AspirazioneSX1,AspirazioneDX2,AspirazioneSX2,CilindroSbloccoRotazione,CilindroSbloccoBascolante);
					TFError(ErrCYLINDER,CilindroSbloccoRotazione^.Status.ErrorID,ADR(CmdExe),ADR(State),ADR(Error),ADR(ErrorLog));
				END_IF

				
			(* Case 100 *)
			100:TFStateUpdate(ADR(State),StateSbloccaRotazione_END);
				TFCommandExeClear(ADR(CmdExe));

			ELSE
				TFError(ErrNOCMDCASE,ErrNULL,ADR(CmdExe),ADR(State),ADR(Error),ADR(ErrorLog));
		END_CASE

		IF TFTimerDone(ADR(Timeout)) THEN
			TFClearAllCmdModulePinzaMagazzino(AspirazioneDX1,AspirazioneSX1,AspirazioneDX2,AspirazioneSX2,CilindroSbloccoRotazione,CilindroSbloccoBascolante);
			TFError(ErrCMDTIMEOUT,ErrNULL,ADR(CmdExe),ADR(State),ADR(Error),ADR(ErrorLog));
		END_IF
		
	(* ******************************************************************************************************** *)
	(* CmdBloccaROTAZIONE - BLOCCA ROTAZIONE *)
	(* ******************************************************************************************************** *)
	CmdBloccaRotazione:
		CASE CmdExe.CmdCase OF
			
			(* Case 0 - Init Command*)
			0: 	TFStateUpdate(ADR(State),StateBloccaRotazione_RUN);
				TFTimerSet(ADR(Timeout),30000+200,TRUE);
				TFTimerSet(ADR(Timer),30000,TRUE);
				IF NOT IN_SimulazioneSenzaHW THEN
					TFCommandCase(ADR(CmdExe),10,CommandCase_JMP);
				ELSE
					TFCommandCase(ADR(CmdExe),100,CommandCase_JMP);
				END_IF
				
			(* Case 10 - CilindroSblocco bacolante *)
			10: 
				CilindroSbloccoRotazione^.Command.Activation 	:= FALSE;
				CilindroSbloccoRotazione^.Command.Deactivation  := TRUE;

				IF (CilindroSbloccoRotazione^.Status.Inactive) THEN
					CilindroSbloccoRotazione^.Command.Activation 	:= FALSE;
					CilindroSbloccoRotazione^.Command.Deactivation := FALSE;
					TFCommandCase(ADR(CmdExe),100,CommandCase_JMP);
				ELSIF CilindroSbloccoBascolante^.Status.ErrorID <> ErrNULL THEN
					TFClearAllCmdModulePinzaMagazzino(AspirazioneDX1,AspirazioneSX1,AspirazioneDX2,AspirazioneSX2,CilindroSbloccoRotazione,CilindroSbloccoBascolante);
					TFError(ErrCYLINDER,CilindroSbloccoBascolante^.Status.ErrorID,ADR(CmdExe),ADR(State),ADR(Error),ADR(ErrorLog));
				END_IF

				
			(* Case 100 *)
			100:TFStateUpdate(ADR(State),StateBloccaBascolante_END);
				TFCommandExeClear(ADR(CmdExe));

			ELSE
				TFError(ErrNOCMDCASE,ErrNULL,ADR(CmdExe),ADR(State),ADR(Error),ADR(ErrorLog));
		END_CASE

		IF TFTimerDone(ADR(Timeout)) THEN
			TFClearAllCmdModulePinzaMagazzino(AspirazioneDX1,AspirazioneSX1,AspirazioneDX2,AspirazioneSX2,CilindroSbloccoRotazione,CilindroSbloccoBascolante);
			TFError(ErrCMDTIMEOUT,ErrNULL,ADR(CmdExe),ADR(State),ADR(Error),ADR(ErrorLog));
		END_IF
		
	(* ******************************************************************************************************** *)
	(* CmdBloccaPinza- BLOCCA ROTAZIONE + BLOCCA BASCULANTE *)
	(* ******************************************************************************************************** *)
	CmdBloccaPinza:
		CASE CmdExe.CmdCase OF
			
			(* Case 0 - Init Command*)
			0: 	TFStateUpdate(ADR(State),StateBloccaPinza_RUN);
				TFTimerSet(ADR(Timeout),30000+200,TRUE);
				TFTimerSet(ADR(Timer),30000,TRUE);
				IF NOT IN_SimulazioneSenzaHW THEN
					TFCommandCase(ADR(CmdExe),10,CommandCase_JMP);
				ELSE
					TFCommandCase(ADR(CmdExe),100,CommandCase_JMP);
				END_IF
				
			(* Case 10 - CilindroSblocco bascolante + rotazione *)
			10: 
				CilindroSbloccoRotazione^.Command.Activation 	:= FALSE;
				CilindroSbloccoRotazione^.Command.Deactivation  := TRUE;
				
				CilindroSbloccoBascolante^.Command.Activation 	:= FALSE;
				CilindroSbloccoBascolante^.Command.Deactivation  := TRUE;

				IF (CilindroSbloccoRotazione^.Status.Inactive) AND CilindroSbloccoRotazione^.Status.Inactive THEN
					CilindroSbloccoRotazione^.Command.Activation 	:= FALSE;
					CilindroSbloccoRotazione^.Command.Deactivation := FALSE;
					CilindroSbloccoBascolante^.Command.Activation 	:= FALSE;
					CilindroSbloccoBascolante^.Command.Deactivation  := FALSE;

					TFCommandCase(ADR(CmdExe),100,CommandCase_JMP);
				ELSIF CilindroSbloccoBascolante^.Status.ErrorID <> ErrNULL THEN
					TFClearAllCmdModulePinzaMagazzino(AspirazioneDX1,AspirazioneSX1,AspirazioneDX2,AspirazioneSX2,CilindroSbloccoRotazione,CilindroSbloccoBascolante);
					TFError(ErrCYLINDER,CilindroSbloccoBascolante^.Status.ErrorID,ADR(CmdExe),ADR(State),ADR(Error),ADR(ErrorLog));
				ELSIF CilindroSbloccoRotazione^.Status.ErrorID <> ErrNULL THEN
					TFClearAllCmdModulePinzaMagazzino(AspirazioneDX1,AspirazioneSX1,AspirazioneDX2,AspirazioneSX2,CilindroSbloccoRotazione,CilindroSbloccoBascolante);
					TFError(ErrCYLINDER,CilindroSbloccoRotazione^.Status.ErrorID,ADR(CmdExe),ADR(State),ADR(Error),ADR(ErrorLog));
				END_IF

				
			(* Case 100 *)
			100:TFStateUpdate(ADR(State),StateBloccaPinza_END);
				TFCommandExeClear(ADR(CmdExe));

			ELSE
				TFError(ErrNOCMDCASE,ErrNULL,ADR(CmdExe),ADR(State),ADR(Error),ADR(ErrorLog));
		END_CASE

		IF TFTimerDone(ADR(Timeout)) THEN
			TFClearAllCmdModulePinzaMagazzino(AspirazioneDX1,AspirazioneSX1,AspirazioneDX2,AspirazioneSX2,CilindroSbloccoRotazione,CilindroSbloccoBascolante);
			TFError(ErrCMDTIMEOUT,ErrNULL,ADR(CmdExe),ADR(State),ADR(Error),ADR(ErrorLog));
		END_IF

	
	(* ******************************************************************************************************** *)
	(* CmdSbloccaPinza- SBLOCCA ROTAZIONE + SBLOCCA BASCULANTE *)
	(* ******************************************************************************************************** *)
	CmdSbloccaPinza:
			CASE CmdExe.CmdCase OF
				
				(* Case 0 - Init Command*)
				0: 	TFStateUpdate(ADR(State),StateSbloccaPinza_RUN);
					TFTimerSet(ADR(Timeout),30000+200,TRUE);
					TFTimerSet(ADR(Timer),30000,TRUE);
					IF NOT IN_SimulazioneSenzaHW THEN
						TFCommandCase(ADR(CmdExe),10,CommandCase_JMP);
					ELSE
						TFCommandCase(ADR(CmdExe),100,CommandCase_JMP);
					END_IF
					
				(* Case 10 - CilindroSblocco bascolante + rotazione *)
				10: 
					CilindroSbloccoBascolante^.Command.Activation 	:= AbilitazioneSbloccoBascolante;
					CilindroSbloccoBascolante^.Command.Deactivation := FALSE;
					CilindroSbloccoRotazione^.Command.Activation 	:= AbilitazioneSbloccoRotazione;
					CilindroSbloccoRotazione^.Command.Deactivation  := FALSE;
	
					IF (CilindroSbloccoBascolante^.Status.Active OR NOT AbilitazioneSbloccoBascolante) AND 
						(CilindroSbloccoRotazione^.Status.Active OR NOT AbilitazioneSbloccoRotazione) THEN
							CilindroSbloccoBascolante^.Command.Activation 	:= FALSE;
							CilindroSbloccoBascolante^.Command.Deactivation := FALSE;
							CilindroSbloccoRotazione^.Command.Activation 	:= FALSE;
							CilindroSbloccoRotazione^.Command.Deactivation  := FALSE;
							TFCommandCase(ADR(CmdExe),100,CommandCase_JMP);
					ELSIF CilindroSbloccoBascolante^.Status.ErrorID <> ErrNULL AND AbilitazioneSbloccoBascolante THEN
						TFClearAllCmdModulePinzaMagazzino(AspirazioneDX1,AspirazioneSX1,AspirazioneDX2,AspirazioneSX2,CilindroSbloccoRotazione,CilindroSbloccoBascolante);
						TFError(ErrCYLINDER,CilindroSbloccoBascolante^.Status.ErrorID,ADR(CmdExe),ADR(State),ADR(Error),ADR(ErrorLog));
					ELSIF CilindroSbloccoRotazione^.Status.ErrorID <> ErrNULL THEN
						TFClearAllCmdModulePinzaMagazzino(AspirazioneDX1,AspirazioneSX1,AspirazioneDX2,AspirazioneSX2,CilindroSbloccoRotazione,CilindroSbloccoBascolante);
						TFError(ErrCYLINDER,CilindroSbloccoRotazione^.Status.ErrorID,ADR(CmdExe),ADR(State),ADR(Error),ADR(ErrorLog));
					END_IF
					
				(* Case 100 *)
				100:TFStateUpdate(ADR(State),StateSbloccaPinza_END);
					TFCommandExeClear(ADR(CmdExe));
	
				ELSE
					TFError(ErrNOCMDCASE,ErrNULL,ADR(CmdExe),ADR(State),ADR(Error),ADR(ErrorLog));
			END_CASE
	
			IF TFTimerDone(ADR(Timeout)) THEN
				TFClearAllCmdModulePinzaMagazzino(AspirazioneDX1,AspirazioneSX1,AspirazioneDX2,AspirazioneSX2,CilindroSbloccoRotazione,CilindroSbloccoBascolante);
				TFError(ErrCMDTIMEOUT,ErrNULL,ADR(CmdExe),ADR(State),ADR(Error),ADR(ErrorLog));
			END_IF
		
	
	(* ******************************************************************************************************** *)
	(* UNLOAD - Attivazione aspirazione + discesa ventose *)
	(* ******************************************************************************************************** *)
	CmdUNLOAD:
		CASE CmdExe.CmdCase OF
			
			(* Case 0 - Init Command*)
			0: 	TFStateUpdate(ADR(State),StateUNLOAD_RUN);
				TFTimerSet(ADR(Timeout),30000+200,TRUE);
				TFTimerSet(ADR(Timer),30000,TRUE);
				DisattivazioneTotaleAspirazioni := FALSE;
				ByPassAttesaDistacco := FALSE;
				IF NOT IN_SimulazioneSenzaHW THEN
					TFCommandCase(ADR(CmdExe),20,CommandCase_JMP);
				ELSE
					TFCommandCase(ADR(CmdExe),100,CommandCase_JMP);
				END_IF
			
			(* Case 20 - Disattivazione aspirazione piastrella *)		
			20: 
				AspirazioneDX1^.Command^.Aspirazione_ON 	:= FALSE;
				AspirazioneDX1^.Command^.Aspirazione_OFF 	:= TRUE;
				AspirazioneSX1^.Command^.Aspirazione_ON 	:= FALSE;
				AspirazioneSX1^.Command^.Aspirazione_OFF 	:= TRUE;
				AspirazioneDX2^.Command^.Aspirazione_ON 	:= FALSE;
				AspirazioneDX2^.Command^.Aspirazione_OFF 	:= TRUE;
				AspirazioneSX2^.Command^.Aspirazione_ON 	:= FALSE;
				AspirazioneSX2^.Command^.Aspirazione_OFF 	:= TRUE;
				IF NOT AspirazioneDX1^.Status.DepressioneSoglia1_OK AND NOT AspirazioneDX1^.Status.DepressioneSoglia1_OK AND
					NOT AspirazioneDX1^.Status.DepressioneSoglia1_OK AND NOT AspirazioneDX1^.Status.DepressioneSoglia1_OK THEN
						ByPassAttesaDistacco := TRUE;
				END_IF
				
				IF AspirazioneDX1^.Status.CommandDone AND AspirazioneSX1^.Status.CommandDone AND
					AspirazioneDX2^.Status.CommandDone AND AspirazioneSX2^.Status.CommandDone THEN
						TFClearAllCmdModulePinzaMagazzino(AspirazioneDX1,AspirazioneSX1,AspirazioneDX2,AspirazioneSX2,CilindroSbloccoRotazione,CilindroSbloccoBascolante);
						StatoPinza.ElementoPrelevato := FALSE;
						TFTimerSet(ADR(TimerAspirazione),HMI_TempoRilascioInDeposito,TRUE);
						TFCommandCase(ADR(CmdExe),30,CommandCase_JMP);
				ELSIF AspirazioneSX1^.Status.ErrorID <> ErrNULL THEN
					TFClearAllCmdModulePinzaMagazzino(AspirazioneDX1,AspirazioneSX1,AspirazioneDX2,AspirazioneSX2,CilindroSbloccoRotazione,CilindroSbloccoBascolante);
					TFError(ErrCYLINDER,AspirazioneSX1^.Status.ErrorID,ADR(CmdExe),ADR(State),ADR(Error),ADR(ErrorLog));
				ELSIF AspirazioneDX1^.Status.ErrorID <> ErrNULL THEN
					TFClearAllCmdModulePinzaMagazzino(AspirazioneDX1,AspirazioneSX1,AspirazioneDX2,AspirazioneSX2,CilindroSbloccoRotazione,CilindroSbloccoBascolante);
					TFError(ErrCYLINDER,AspirazioneDX1^.Status.ErrorID,ADR(CmdExe),ADR(State),ADR(Error),ADR(ErrorLog));
				END_IF
			
			(* Case 30 - Attesa tempo distacco *)		
			30:
				IF TFTimerDone(ADR(TimerAspirazione)) OR ByPassAttesaDistacco THEN
					IF IN.RichiestaRicalibrazioneOvemEsterna THEN
						IN.RichiestaRicalibrazioneOvemEsterna := FALSE;
						TFCommandCase(ADR(CmdExe),40,CommandCase_JMP);
					ELSE
						TFCommandCase(ADR(CmdExe),100,CommandCase_JMP);
					END_IF		
				END_IF
				
			(* Case 40 - Attesa tempo distacco *)		
			40:	
				AspirazioneDX1^.Command^.Aspirazione_ON_ScritturaSoglia 	:= TRUE;
				AspirazioneSX1^.Command^.Aspirazione_ON_ScritturaSoglia 	:= TRUE;
				AspirazioneDX2^.Command^.Aspirazione_ON_ScritturaSoglia 	:= TRUE;
				AspirazioneSX2^.Command^.Aspirazione_ON_ScritturaSoglia 	:= TRUE;
				IF AspirazioneDX1^.Status.CommandDone AND AspirazioneSX1^.Status.CommandDone AND
					AspirazioneDX2^.Status.CommandDone AND AspirazioneSX2^.Status.CommandDone THEN
						TFClearAllCmdModulePinzaMagazzino(AspirazioneDX1,AspirazioneSX1,AspirazioneDX2,AspirazioneSX2,CilindroSbloccoRotazione,CilindroSbloccoBascolante);
						TFCommandCase(ADR(CmdExe),100,CommandCase_JMP);
				ELSIF TFTimerDone(ADR(Timer)) THEN
					TFClearAllCmdModulePinzaMagazzino(AspirazioneDX1,AspirazioneSX1,AspirazioneDX2,AspirazioneSX2,CilindroSbloccoRotazione,CilindroSbloccoBascolante);
					TFError(ErrTOHOME,ErrNULL,ADR(CmdExe),ADR(State),ADR(Error),ADR(ErrorLog));
				END_IF
				
			(* Case 100 *)
			100:
				StatoPinza.ElementoPrelevato := FALSE;
				TFStateUpdate(ADR(State),StateUNLOAD_END);
				TFCommandExeClear(ADR(CmdExe));

			ELSE
				TFError(ErrNOCMDCASE,ErrNULL,ADR(CmdExe),ADR(State),ADR(Error),ADR(ErrorLog));
		END_CASE

		IF TFTimerDone(ADR(Timeout)) THEN
			TFClearAllCmdModulePinzaMagazzino(AspirazioneDX1,AspirazioneSX1,AspirazioneDX2,AspirazioneSX2,CilindroSbloccoRotazione,CilindroSbloccoBascolante);
			TFError(ErrCMDTIMEOUT,ErrNULL,ADR(CmdExe),ADR(State),ADR(Error),ADR(ErrorLog));
		END_IF

	(* ******************************************************************************************************** *)
	(* POSTUNLOAD - AGGANCIO BASCULANTE *)
	(* ******************************************************************************************************** *)
	CmdPOSTUNLOAD:
		CASE CmdExe.CmdCase OF
			
			(* Case 0 - Init Command*)
			0: 	TFStateUpdate(ADR(State),StatePOSTUNLOAD_RUN);
				TFTimerSet(ADR(Timeout),30000+200,TRUE);
				TFTimerSet(ADR(Timer),30000,TRUE);
				IF NOT IN_SimulazioneSenzaHW THEN
					TFCommandCase(ADR(CmdExe),10,CommandCase_JMP);
				ELSE
					TFCommandCase(ADR(CmdExe),100,CommandCase_JMP);
				END_IF
				
			(* Case 10 - CilindroSbloccoRotazione *)
			10: 
				CilindroSbloccoRotazione^.Command.Activation 	:= FALSE;
				CilindroSbloccoRotazione^.Command.Deactivation 	:= TRUE;

				IF (CilindroSbloccoRotazione^.Status.Inactive)THEN
					CilindroSbloccoRotazione^.Command.Activation 	:= FALSE;
					CilindroSbloccoRotazione^.Command.Deactivation 	:= FALSE;
					TFCommandCase(ADR(CmdExe),100,CommandCase_JMP);
				ELSIF CilindroSbloccoRotazione^.Status.ErrorID <> ErrNULL THEN
					TFClearAllCmdModulePinzaMagazzino(AspirazioneDX1,AspirazioneSX1,AspirazioneDX2,AspirazioneSX2,CilindroSbloccoRotazione,CilindroSbloccoBascolante);
					TFError(ErrCYLINDER,CilindroSbloccoRotazione^.Status.ErrorID,ADR(CmdExe),ADR(State),ADR(Error),ADR(ErrorLog));
				END_IF
			
			(* Case 100 *)
			100:TFStateUpdate(ADR(State),StatePOSTUNLOAD_END);
				TFCommandExeClear(ADR(CmdExe));

			ELSE
				TFError(ErrNOCMDCASE,ErrNULL,ADR(CmdExe),ADR(State),ADR(Error),ADR(ErrorLog));
		END_CASE

		IF TFTimerDone(ADR(Timeout)) THEN
			TFClearAllCmdModulePinzaMagazzino(AspirazioneDX1,AspirazioneSX1,AspirazioneDX2,AspirazioneSX2,CilindroSbloccoRotazione,CilindroSbloccoBascolante);
			TFError(ErrCMDTIMEOUT,ErrNULL,ADR(CmdExe),ADR(State),ADR(Error),ADR(ErrorLog));
		END_IF

	ELSE
		TFError(ErrNOCMD,ErrNULL,ADR(CmdExe),ADR(State),ADR(Error),ADR(ErrorLog));

END_CASE;


(* ******************************************************************************************************** *)
(* State Input/Output *)
(* ******************************************************************************************************** *)
(* Fill Input/Output bit with sensor, electrovalve, etc. status *)

StatoPinza.LatoDxPiastrellaInPresa	:= ((AspirazioneDX1^.Status.DepressioneSoglia1_OK AND AspirazioneDX2^.Status.DepressioneSoglia1_OK)  OR IN.ByPassSensoreVuoto);// AND NOT IN.TastoreCartoneDX;
StatoPinza.LatoSxPiastrellaInPresa	:=((AspirazioneSX1^.Status.DepressioneSoglia1_OK AND AspirazioneSX2^.Status.DepressioneSoglia1_OK)  OR IN.ByPassSensoreVuoto);// AND NOT IN.TastoreCartoneSX;
StatoPinza.RotazioneBloccata		:= CilindroSbloccoRotazione^.Status.Inactive;
StatoPinza.RotazioneSbloccata 		:= CilindroSbloccoRotazione^.Status.Active;
StatoPinza.PianoInPresa				:= StatoPinza.LatoDxPiastrellaInPresa AND StatoPinza.LatoSxPiastrellaInPresa OR (IN.ByPassSensoreVuoto AND StatoPinza.ElementoPrelevato);

(* ******************************************************************************************************** *)
(* Input *)
(* ******************************************************************************************************** *)

(* ******************************************************************************************************** *)
(* Alarm *)
(* ******************************************************************************************************** *)

(* ******************************************************************************************************** *)
(* Error Check - Clear All Output!!! *)
(* ******************************************************************************************************** *)
IF Error.Code > ErrNULL THEN
	IF CmdExe.Code <> CmdNOP THEN
		IF CmdExe.Code <> CmdSTOP AND
			CmdExe.Code <> CmdPOWER AND
			CmdExe.Code <> CmdRESET AND
			CmdExe.Code <> CmdMAN AND
			CmdExe.Code <> CmdLOAD AND
			CmdExe.Code <> CmdUNLOAD THEN
			TFCommandClear(ADR(CmdNext));
			TFCommandExeClear(ADR(CmdExe));

			(* Clear All Output Here *)

		END_IF;
	END_IF;
END_IF;


(* ******************************************************************************************************** *)
(* Common Outputs *)
(* ******************************************************************************************************** *)

END_FUNCTION_BLOCK

(* stored: Version 1.1.0.1, ProductVersion 3.1.4024.11
   POU TFModulePalletizer_Pinza_mag: Id {a01c6770-8d6e-40a0-84eb-4ca0b2b11347}, SpecialFunc None *)
